Staubli VAL3: isBinary.pgx

program isBinary(string x_sBinary, bool& x_bRes)
  local num l_nIndex
begin

  for l_nIndex= 0 to len(x_sBinary)-1
    if mid(x_sBinary, 1, l_nIndex)!="0" and mid(x_sBinary, 1, l_nIndex)!="1"
      x_bRes = false
      return
    endIf
  endFor

  x_bRes = true

end
